RoboDK station: Estacion2.rdk

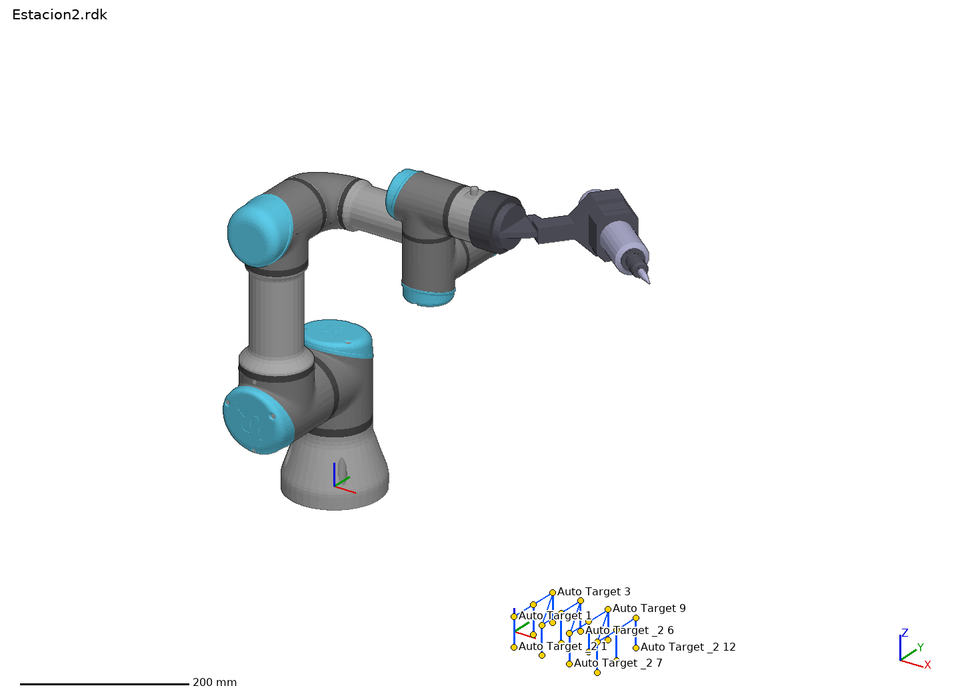
[picture v0: the station drawn from its stored meshes, robots at their saved joint values, targets as dots, program paths as lines]
Station Estacion2 (saved by RoboDK 5.6.0). Poses are relative to the parent item; angles as X-Y-Z fixed-axis rotations.
  - frame UR3 Base at (0, 0, 0) mm
    - robot UR3: 6 axes, payload 3 kg, reach 500 mm, repeatability 0.1 mm, weight 11 kg
        modified DH rows (alpha deg, a mm, theta deg, d mm): 0, 0, 0, 151.9; 90, 0, 180, 0; 0, 243.65, 0, 0; 0, 213, 0, 110.4; -90, 0, 0, 83.4; 90, 0, 180, 82.4
        joint limits [-360, -360, -360, -360, -360, -360] to [360, 360, 360, 360, 360, 360]; home [0, -90, -90, 0, 90, 0]; saved at [0, -90, -90, 0, 90, 0]
      - tool Spintech Spindle, TCP at (32, 0, 260) mm, rotated rx 0 ry 39 rz 0 deg, size 157.3 x 72 x 259.9 mm
  - frame Frame1 at (400, -200, 0) mm
    - target Auto Target 1 (Cartesian target) at (0, 0, 20) mm, rotated rx -180 ry 0 rz 180 deg; joints [113.901, -87.825, 120.548, 219.113, -54.876, 29.694] of UR3
    - target Auto Target _2 1 (Cartesian target) at (0, 0, -20) mm, rotated rx -180 ry 0 rz 180 deg; joints [113.901, -80.706, 126.282, 206.26, -54.876, 29.694] of UR3
    - target Auto Target 2 (Cartesian target) at (0, 40, 20) mm, rotated rx -180 ry 0 rz 180 deg; joints [117.848, -93.729, 127.47, 215.539, -56.19, 34.208] of UR3
    - target Auto Target _2 2 (Cartesian target) at (0, 40, -20) mm, rotated rx -180 ry 0 rz 180 deg; joints [117.848, -85.632, 133.562, 201.349, -56.19, 34.208] of UR3
    - target Auto Target 3 (Cartesian target) at (0, 80, 20) mm, rotated rx -180 ry 0 rz 180 deg; joints [122.96, -98.899, 133.191, 211.93, -58.128, 39.841] of UR3
    - target Auto Target _2 3 (Cartesian target) at (0, 80, -20) mm, rotated rx -180 ry 0 rz 180 deg; joints [122.96, -89.741, 139.646, 196.318, -58.128, 39.841] of UR3
    - target Auto Target 4 (Cartesian target) at (40, 0, 20) mm, rotated rx -180 ry 0 rz 180 deg; joints [121.069, -79.302, 112.698, 213.924, -57.382, 37.785] of UR3
    - target Auto Target _2 4 (Cartesian target) at (40, 0, -20) mm, rotated rx -180 ry 0 rz 180 deg; joints [121.069, -72.732, 117.686, 202.366, -57.382, 37.785] of UR3
    - target Auto Target 5 (Cartesian target) at (40, 40, 20) mm, rotated rx -180 ry 0 rz 180 deg; joints [125.442, -83.908, 119.309, 209.446, -59.155, 42.485] of UR3
    - target Auto Target _2 5 (Cartesian target) at (40, 40, -20) mm, rotated rx -180 ry 0 rz 180 deg; joints [125.442, -76.541, 124.454, 196.933, -59.155, 42.485] of UR3
    - target Auto Target 6 (Cartesian target) at (40, 80, 20) mm, rotated rx -180 ry 0 rz 180 deg; joints [130.795, -87.67, 124.647, 205.141, -61.547, 47.997] of UR3
    - target Auto Target _2 6 (Cartesian target) at (40, 80, -20) mm, rotated rx -180 ry 0 rz 180 deg; joints [130.795, -79.492, 129.941, 191.67, -61.547, 47.997] of UR3
    - target Auto Target 7 (Cartesian target) at (80, 0, 20) mm, rotated rx -180 ry 0 rz 180 deg; joints [127.061, -71.218, 103.233, 211.971, -59.855, 44.18] of UR3
    - target Auto Target _2 7 (Cartesian target) at (80, 0, -20) mm, rotated rx -180 ry 0 rz 180 deg; joints [127.061, -65.313, 107.713, 201.586, -59.855, 44.18] of UR3
    - target Auto Target 8 (Cartesian target) at (80, 40, 20) mm, rotated rx -180 ry 0 rz 180 deg; joints [131.559, -75.099, 109.581, 207.273, -61.907, 48.763] of UR3
    - target Auto Target _2 8 (Cartesian target) at (80, 40, -20) mm, rotated rx -180 ry 0 rz 180 deg; joints [131.559, -68.582, 114.095, 196.241, -61.907, 48.763] of UR3
    - target Auto Target 9 (Cartesian target) at (80, 80, 20) mm, rotated rx -180 ry 0 rz 180 deg; joints [136.844, -78.148, 114.596, 202.981, -64.504, 53.92] of UR3
    - target Auto Target _2 9 (Cartesian target) at (80, 80, -20) mm, rotated rx -180 ry 0 rz 180 deg; joints [136.844, -71.05, 119.147, 191.331, -64.504, 53.92] of UR3
    - target Auto Target 10 (Cartesian target) at (120, 0, 20) mm, rotated rx -180 ry 0 rz 180 deg; joints [132.087, -63.289, 92.239, 212.559, -62.158, 49.288] of UR3
    - target Auto Target _2 10 (Cartesian target) at (120, 0, -20) mm, rotated rx -180 ry 0 rz 180 deg; joints [132.087, -58.059, 96.427, 203.141, -62.158, 49.288] of UR3
    - target Auto Target 11 (Cartesian target) at (120, 40, 20) mm, rotated rx -180 ry 0 rz 180 deg; joints [136.545, -66.796, 98.479, 207.868, -64.352, 53.635] of UR3
    - target Auto Target _2 11 (Cartesian target) at (120, 40, -20) mm, rotated rx -180 ry 0 rz 180 deg; joints [136.545, -61.088, 102.615, 198.024, -64.352, 53.635] of UR3
    - target Auto Target 12 (Cartesian target) at (120, 80, 20) mm, rotated rx -180 ry 0 rz 180 deg; joints [141.627, -69.489, 103.314, 203.765, -67.004, 58.393] of UR3
    - target Auto Target _2 12 (Cartesian target) at (120, 80, -20) mm, rotated rx -180 ry 0 rz 180 deg; joints [141.627, -63.354, 107.42, 193.524, -67.004, 58.393] of UR3
  - Python program Prog1 (listed below)
  - program AutoProgram (36 instructions, listed below)
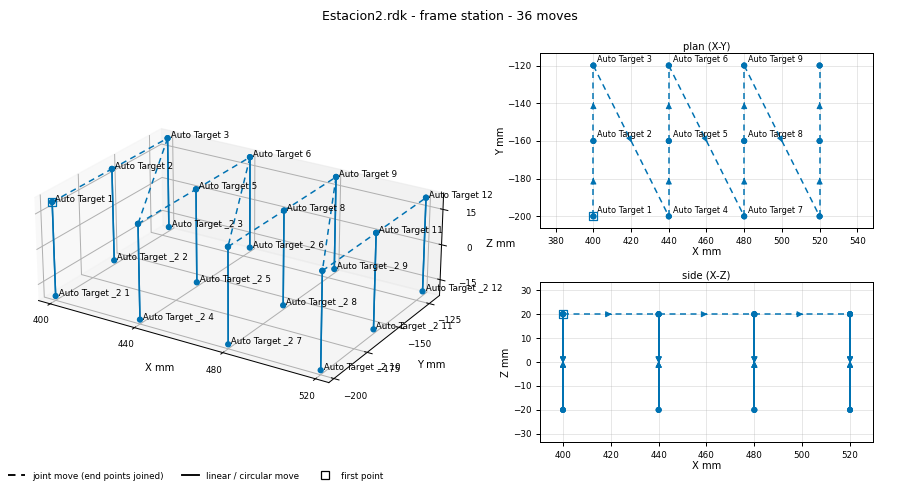
[picture p0: tool path of Estacion2.rdk in frame station, 36 of 36 moves have a stored position in this frame; points joined in program order, loops and branches not executed]

--- Python program Prog1 ---
# Type help("robodk.robolink") or help("robodk.robomath") for more information
# Press F5 to run the script
# Documentation: https://robodk.com/doc/en/RoboDK-API.html
# Reference:     https://robodk.com/doc/en/PythonAPI/robodk.html
# Note: It is not required to keep a copy of this file, your Python script is saved with your RDK project

# You can also use the new version of the API:
from robodk.robolink import *
from robodk.robomath import *

def gridXY(m, n, d):
    listaPuntos = []
    for i in range(m):
        for j in range(n):
            punto = [i*d, j*d, 20]
            listaPuntos.append(punto)

    return listaPuntos

m = 4
n = 3
d = 40

puntos = gridXY(m, n, d)

RDK = Robolink()
#pose = eye()

list_names = RDK.ItemList(None, True)

for item_name in list_names:
    if item_name.startswith('Auto'):
        RDK.Item(item_name).Delete()

myRobot = RDK.Item('UR3', ITEM_TYPE_ROBOT)

myFrame = RDK.Item("Frame1")

myRobot.setPoseFrame(myFrame)

pose_ref = myRobot.Pose()

pose_k = pose_ref

# Creamos un Programa
prog = RDK.AddProgram("AutoProgram")
j = 0

for i in puntos:
    # Target
    ti = RDK.AddTarget("Auto Target %i" % (j+1))
    pose_i = pose_ref
    pose_i.setPos(i)
    ti.setPose(pose_i)
    ti.setAsCartesianTarget()
    ti.setVisible(0)
    prog.MoveJ(ti)

    ti2 = RDK.AddTarget("Auto Target _2 %i" % (j+1))
    pose_j = pose_i
    pose_j.setPos([i[0], i[1], -20])
    ti2.setPose(pose_j)
    ti2.setAsCartesianTarget()
    ti2.setVisible(0)
    prog.MoveL(ti2)
    pose_i.setPos(i)
    prog.MoveL(ti)
    j +=1


print("DONE")

--- program AutoProgram (robot UR3) ---
  MoveJ (Auto Target 1)
  MoveL (Auto Target _2 1)
  MoveL (Auto Target 1)
  MoveJ (Auto Target 2)
  MoveL (Auto Target _2 2)
  MoveL (Auto Target 2)
  MoveJ (Auto Target 3)
  MoveL (Auto Target _2 3)
  MoveL (Auto Target 3)
  MoveJ (Auto Target 4)
  MoveL (Auto Target _2 4)
  MoveL (Auto Target 4)
  MoveJ (Auto Target 5)
  MoveL (Auto Target _2 5)
  MoveL (Auto Target 5)
  MoveJ (Auto Target 6)
  MoveL (Auto Target _2 6)
  MoveL (Auto Target 6)
  MoveJ (Auto Target 7)
  MoveL (Auto Target _2 7)
  MoveL (Auto Target 7)
  MoveJ (Auto Target 8)
  MoveL (Auto Target _2 8)
  MoveL (Auto Target 8)
  MoveJ (Auto Target 9)
  MoveL (Auto Target _2 9)
  MoveL (Auto Target 9)
  MoveJ (Auto Target 10)
  MoveL (Auto Target _2 10)
  MoveL (Auto Target 10)
  MoveJ (Auto Target 11)
  MoveL (Auto Target _2 11)
  MoveL (Auto Target 11)
  MoveJ (Auto Target 12)
  MoveL (Auto Target _2 12)
  MoveL (Auto Target 12)
